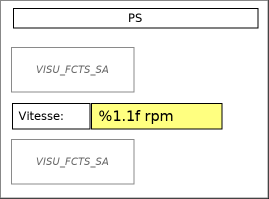
VISUALIZATION SA_PS  // 269x199
    Rectangle (0,0 269x199)
    Rectangle (12,103 78x26), "Vitesse:"
    Rectangle (13,8 245x20), "PS"
    Rectangle (91,103 131x26), "%1.1f rpm", text variable: PRG_MOUVEMENT_PS.ROTATION_PS.PRM_Vitesse, input disabled if: ((NOT PRG_User.ACTU_USER.MAINTENANCE AND NOT PRG_User.ACTU_USER.FONCTION_SA AND NOT PRG_User.ACTU_USER.MODIF_ENLIGNE) OR (NOT MACHINE.STATE_Wait_Prod AND NOT MACHINE.STATE_Manu)) <> 0
        OnMouseDown: write the text variable via InputWithLimits, min 0.2, max 20.0
    Frame (11,47 123x45)
        shows VISU_FCTS_SA(m_Input_ID_XML := 15, m_Input_UserRight := PRG_USER.ACTU_USER.FONCTION_SA, m_Input_Operation := PRG_MOUVEMENT_PS.ROTATION_PS.OP_Rotation)
    Frame (11,139 123x45)
        shows VISU_FCTS_SA(m_Input_ID_XML := 7, m_Input_UserRight := PRG_USER.ACTU_USER.FONCTION_SA, m_Input_Operation := PRG_MOUVEMENT_PS.ROTATION_PS.OP_Stop)
END_VISUALIZATION

(* stored: Version 1.1.0.1, ProductVersion 3.1.4024.12
   Visu SA_PS: Id {846640be-cfe1-46a8-bbe4-545fa19046a1} *)
